FUNCTION_BLOCK pHTank
  (* Standard: 61499-2 *)
  (* Version 0.1, 2015-00-13, Th?o, PC_THEO *)
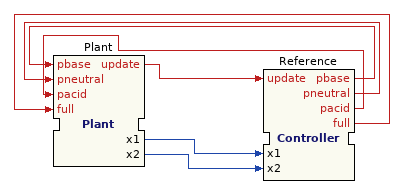
  FBS
    Plant : Plant;
    Reference : Controller;
  END_FBS
  EVENT_CONNECTIONS
    Plant.update TO Reference.update;
    Reference.pbase TO Plant.pbase;
    Reference.pneutral TO Plant.pneutral;
    Reference.pacid TO Plant.pacid;
    Reference.full TO Plant.full;
  END_CONNECTIONS
  DATA_CONNECTIONS
    Plant.x1 TO Reference.x1;
    Plant.x2 TO Reference.x2;
  END_CONNECTIONS
END_FUNCTION_BLOCK
